// TwinCAT 3 PLC project virtual_plc
// ProgramVersion: 3.1.4024.0
// libraries:
//   Tc2_Standard, * (Beckhoff Automation GmbH)
//   Tc2_System, * (Beckhoff Automation GmbH)
//   Tc3_Module, * (Beckhoff Automation GmbH)
// project tree:
//   GVLs/ GVL_MorningRoutine.TcGVL
//   / PlcTask.TcTTO
//   POUs/ MAIN.TcPOU, IsReady.TcPOU, PRG_BreakfastTask.TcPOU, PRG_WakeUpTask.TcPOU
// real-time tasks:
//   TASK PlcTask: cycle T#50000us, priority 20, ADS port 350

CONFIGURATION virtual_plc
    RESOURCE PLC ON TwinCAT3
        TASK PlcTask(INTERVAL := T#50000us, PRIORITY := 20);
        PROGRAM MAIN WITH PlcTask : MAIN;
        PROGRAM PRG_BreakfastTask WITH PlcTask : PRG_BreakfastTask;
        PROGRAM PRG_WakeUpTask WITH PlcTask : PRG_WakeUpTask;
    END_RESOURCE
END_CONFIGURATION

// ---- GVLs/GVL_MorningRoutine.TcGVL
{attribute 'qualified_only'}
VAR_GLOBAL
	// Task 1 — Wake Up Routine
    AlarmOn : BOOL := FALSE;
    GotOutOfBed : BOOL := FALSE;
    BrushedTeeth : BOOL := FALSE;
    ReadyForBreakfast : BOOL := FALSE;
    State_WakeUp : INT := 0;
    StartWakeUp : BOOL := TRUE;

    // Task 2 — Breakfast Routine
    MakingBreakfast : BOOL := FALSE;
    EatingBreakfast : BOOL := FALSE;
    ReadyToLeave : BOOL := FALSE;
    State_Breakfast : INT := 0;
    StartBreakfast : BOOL := TRUE;
END_VAR

// ---- POUs/MAIN.TcPOU
PROGRAM MAIN
VAR
END_VAR

END_PROGRAM

// ---- POUs/PRG_BreakfastTask.TcPOU
PROGRAM PRG_BreakfastTask
VAR
	Ready : BOOL;
END_VAR

CASE GVL_MorningRoutine.State_Breakfast OF

    0: // Idle
        IF GVL_MorningRoutine.StartBreakfast THEN
            GVL_MorningRoutine.State_Breakfast := 10;
        END_IF

    10: // Wait for Task 1 to finish
        Ready := IsReady(GVL_MorningRoutine.ReadyForBreakfast);
        IF Ready THEN
            GVL_MorningRoutine.State_Breakfast := 20;
        END_IF

    20: // Make breakfast
        GVL_MorningRoutine.MakingBreakfast := TRUE;
        GVL_MorningRoutine.State_Breakfast := 30;

    30: // Eat breakfast
        GVL_MorningRoutine.EatingBreakfast := TRUE;
        GVL_MorningRoutine.ReadyToLeave := TRUE;
        GVL_MorningRoutine.State_Breakfast := 40;

    40: // Done
        // Task completed

END_CASE

END_PROGRAM

// ---- POUs/IsReady.TcPOU
FUNCTION IsReady : BOOL
VAR_INPUT
	Condition : BOOL;
END_VAR

IsReady := Condition;

END_FUNCTION

// ---- POUs/PRG_WakeUpTask.TcPOU
PROGRAM PRG_WakeUpTask
VAR
END_VAR

CASE GVL_MorningRoutine.State_WakeUp OF

    0: // Idle
        IF GVL_MorningRoutine.StartWakeUp THEN
            GVL_MorningRoutine.AlarmOn := TRUE;
            GVL_MorningRoutine.State_WakeUp := 10;
        END_IF

    10: // Alarm is ringing
        // Simulate waking up
        GVL_MorningRoutine.GotOutOfBed := TRUE;
        GVL_MorningRoutine.State_WakeUp := 20;

    20: // Brush teeth
        GVL_MorningRoutine.BrushedTeeth := TRUE;
        GVL_MorningRoutine.ReadyForBreakfast := TRUE;
        GVL_MorningRoutine.State_WakeUp := 30;

    30: // Done
        // Task finished, no further action

END_CASE

END_PROGRAM
